Fanuc KAREL source: kb00157.KL

PROGRAM KB00157
%STACKSIZE=65535
%PRIORITY=65535
%NOLOCKGROUP
VAR
P1 : INTEGER
RESULT : INTEGER
BEGIN
P1=1
RESULT=SEMA_COUNT(P1)
END KB00157
